// This function has been automatically generated from the project information.
{attribute 'signature_flag' := '1073741824'}
{attribute 'TcGenerated'}
{attribute 'no-analysis'}
FUNCTION F_GetCompany : WSTRING
VAR_INPUT
	
END_VAR

F_GetCompany := "Beckhoff Automation Belgium";

END_FUNCTION

(* stored: Version 1.1.0.1
   POU F_GetCompany: Id {c4cacaf6-de54-491b-aa30-40f2b1b7af6d}, SpecialFunc None *)
